SUBAPPLICATION Uebung_006c (* SR-Flip-Flop mit IB auf DI_REPEAT *)
  (* Standard: 61499-2; Description: Copyright (c) 2023 Meisterschulen am Ostbahnhof This program and the accompanying materials are made available under the terms of the Eclipse Public License 2.0 which is available at https://www.eclipse.org/legal/epl-2.0/ SPDX-License-Identifier: EPL-2.0 *)
  (* Version 1.0, 2023-10-23, Franz Höpfinger, Meisterschulen am Ostbahnhof *)
  PACKAGE Uebungen;
  IMPORT logiBUS::io::DI::logiBUS_DI::Input_I1;
  IMPORT logiBUS::io::DI::logiBUS_DI::Input_I2;
  IMPORT logiBUS::io::DI::logiBUS_DI_Events::BUTTON_PRESS_REPEAT;
  IMPORT logiBUS::io::DQ::logiBUS_DO::Output_Q1;
  IMPORT logiBUS::io::DQ::logiBUS_DO::Output_Q2;
  IMPORT logiBUS::io::DQ::logiBUS_DO::Output_Q3;
  IMPORT logiBUS::io::DQ::logiBUS_DO::Output_Q4;
  IMPORT logiBUS::io::DQ::logiBUS_DO::Output_Q5;
  IMPORT logiBUS::io::DQ::logiBUS_DO::Output_Q6;
  IMPORT logiBUS::io::DQ::logiBUS_DO::Output_Q7;
  IMPORT logiBUS::io::DQ::logiBUS_DO::Output_Q8;
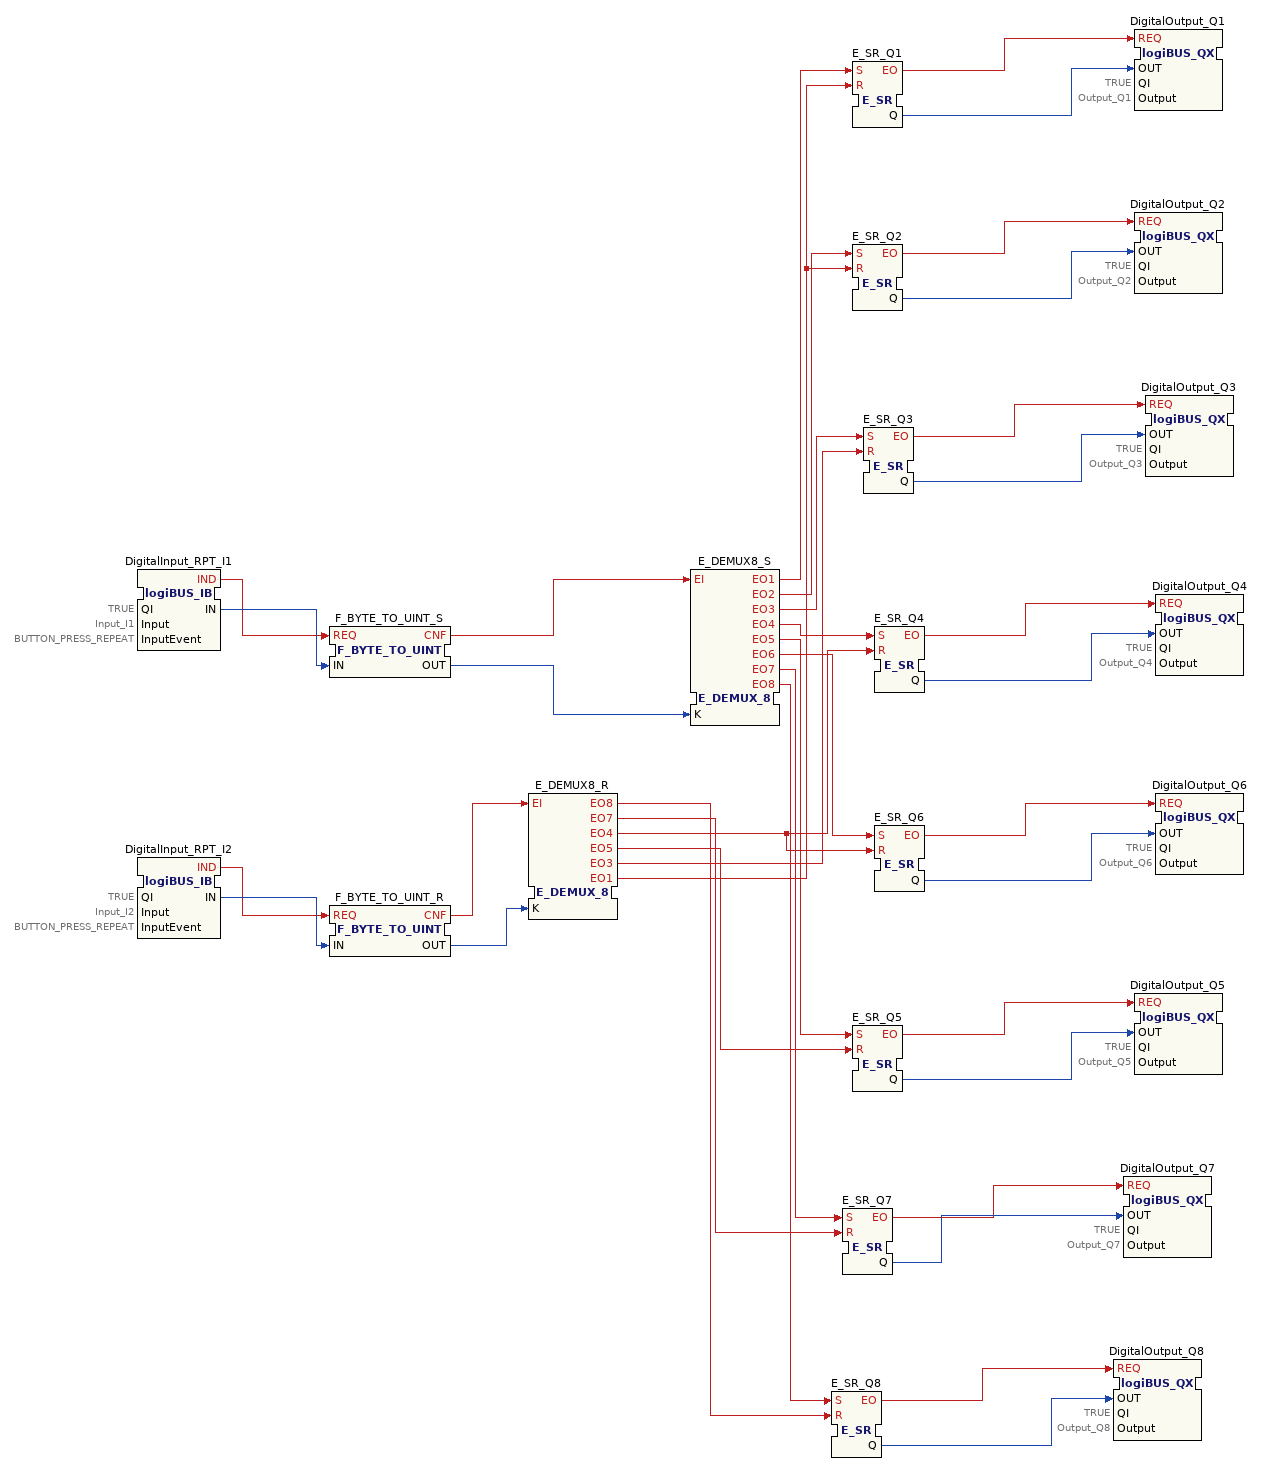
  FBS
    DigitalOutput_Q1 : logiBUS::io::DQ::logiBUS_QX(QI := TRUE, Output := Output_Q1);
    DigitalInput_RPT_I1 : logiBUS::io::DI::logiBUS_IB(QI := TRUE, Input := Input_I1, InputEvent := BUTTON_PRESS_REPEAT);
    DigitalInput_RPT_I2 : logiBUS::io::DI::logiBUS_IB(QI := TRUE, Input := Input_I2, InputEvent := BUTTON_PRESS_REPEAT);
    E_SR_Q1 : iec61499::events::E_SR;
    E_SR_Q2 : iec61499::events::E_SR;
    DigitalOutput_Q2 : logiBUS::io::DQ::logiBUS_QX(QI := TRUE, Output := Output_Q2);
    DigitalOutput_Q3 : logiBUS::io::DQ::logiBUS_QX(QI := TRUE, Output := Output_Q3);
    DigitalOutput_Q4 : logiBUS::io::DQ::logiBUS_QX(QI := TRUE, Output := Output_Q4);
    E_SR_Q5 : iec61499::events::E_SR;
    E_SR_Q6 : iec61499::events::E_SR;
    DigitalOutput_Q5 : logiBUS::io::DQ::logiBUS_QX(QI := TRUE, Output := Output_Q5);
    DigitalOutput_Q6 : logiBUS::io::DQ::logiBUS_QX(QI := TRUE, Output := Output_Q6);
    DigitalOutput_Q7 : logiBUS::io::DQ::logiBUS_QX(QI := TRUE, Output := Output_Q7);
    DigitalOutput_Q8 : logiBUS::io::DQ::logiBUS_QX(QI := TRUE, Output := Output_Q8);
    E_DEMUX8_S : iec61499::events::E_DEMUX_8;
    E_DEMUX8_R : iec61499::events::E_DEMUX_8;
    E_SR_Q3 : iec61499::events::E_SR;
    E_SR_Q4 : iec61499::events::E_SR;
    E_SR_Q7 : iec61499::events::E_SR;
    E_SR_Q8 : iec61499::events::E_SR;
    F_BYTE_TO_UINT_S : iec61131::conversion::F_BYTE_TO_UINT;
    F_BYTE_TO_UINT_R : iec61131::conversion::F_BYTE_TO_UINT;
  END_FBS
  EVENT_CONNECTIONS
    E_SR_Q1.EO TO DigitalOutput_Q1.REQ;
    E_SR_Q2.EO TO DigitalOutput_Q2.REQ;
    E_SR_Q5.EO TO DigitalOutput_Q5.REQ;
    E_DEMUX8_S.EO1 TO E_SR_Q1.S;
    E_SR_Q4.EO TO DigitalOutput_Q4.REQ;
    E_SR_Q3.EO TO DigitalOutput_Q3.REQ;
    E_DEMUX8_S.EO2 TO E_SR_Q2.S;
    E_DEMUX8_S.EO3 TO E_SR_Q3.S;
    E_DEMUX8_S.EO4 TO E_SR_Q4.S;
    E_DEMUX8_S.EO5 TO E_SR_Q5.S;
    E_SR_Q6.EO TO DigitalOutput_Q6.REQ;
    E_SR_Q8.EO TO DigitalOutput_Q8.REQ;
    E_SR_Q7.EO TO DigitalOutput_Q7.REQ;
    E_DEMUX8_S.EO6 TO E_SR_Q6.S;
    E_DEMUX8_S.EO7 TO E_SR_Q7.S;
    E_DEMUX8_S.EO8 TO E_SR_Q8.S;
    F_BYTE_TO_UINT_S.CNF TO E_DEMUX8_S.EI;
    DigitalInput_RPT_I1.IND TO F_BYTE_TO_UINT_S.REQ;
    DigitalInput_RPT_I2.IND TO F_BYTE_TO_UINT_R.REQ;
    F_BYTE_TO_UINT_R.CNF TO E_DEMUX8_R.EI;
    E_DEMUX8_R.EO8 TO E_SR_Q8.R;
    E_DEMUX8_R.EO7 TO E_SR_Q7.R;
    E_DEMUX8_R.EO4 TO E_SR_Q6.R;
    E_DEMUX8_R.EO5 TO E_SR_Q5.R;
    E_DEMUX8_R.EO4 TO E_SR_Q4.R;
    E_DEMUX8_R.EO3 TO E_SR_Q3.R;
    E_DEMUX8_R.EO1 TO E_SR_Q2.R;
    E_DEMUX8_R.EO1 TO E_SR_Q1.R;
  END_CONNECTIONS
  DATA_CONNECTIONS
    E_SR_Q1.Q TO DigitalOutput_Q1.OUT;
    E_SR_Q2.Q TO DigitalOutput_Q2.OUT;
    E_SR_Q5.Q TO DigitalOutput_Q5.OUT;
    E_SR_Q3.Q TO DigitalOutput_Q3.OUT;
    E_SR_Q4.Q TO DigitalOutput_Q4.OUT;
    E_SR_Q6.Q TO DigitalOutput_Q6.OUT;
    E_SR_Q8.Q TO DigitalOutput_Q8.OUT;
    E_SR_Q7.Q TO DigitalOutput_Q7.OUT;
    F_BYTE_TO_UINT_S.OUT TO E_DEMUX8_S.K;
    DigitalInput_RPT_I1.IN TO F_BYTE_TO_UINT_S.IN;
    DigitalInput_RPT_I2.IN TO F_BYTE_TO_UINT_R.IN;
    F_BYTE_TO_UINT_R.OUT TO E_DEMUX8_R.K;
  END_CONNECTIONS
END_SUBAPPLICATION
